// TIA Portal V16 export
// export: Created 2024-09-05T17:40:14.2049484Z, ExportSetting WithDefaults, DisplayName Totally Integrated Automation Portal, DisplayVersion V16 Update 6, DisplayName TIA Portal Version Control Interface, DisplayVersion V16 Update 2, DisplayName TIA Portal Openness, DisplayVersion V16 Update 6, DisplayName STEP 7 Professional, DisplayVersion V16 Update 6, DisplayName STEP 7 Safety, DisplayVersion V16, DisplayName WinCC Advanced, DisplayVersion V16 Update 6
TYPE "UDT_TurnTableCommands"
// stored: IsFailsafeCompliant false
   STRUCT
      ReadyToJogCW : Bool;
      JogCW : Bool;
      ReadyToJogCCW : Bool;
      JogCCW : Bool;
      ReadyToStartCW : Bool;
      StartCW : Bool;
      ReadyToStartCCW : Bool;
      StartCCW : Bool;
   END_STRUCT;
END_TYPE
